{attribute 'qualified_only'}
VAR_GLOBAL
	GC : ARRAY[1..Param_Config.MaxModulePerType] OF FB_GC_Module;
	GC_Runtime : ARRAY[1..Param_Config.MaxModulePerType] OF ST_ModuleRuntimeConfig;
	GC_Control : ARRAY[1..Param_Config.MaxModulePerType] OF ST_GC_CtrlStatus;
	GC_SpinAxis : ARRAY[1..Param_Config.MaxModulePerType] OF I_Axis_BaseUnit;
	GC_LiftPinAxis : ARRAY[1..Param_Config.MaxModulePerType] OF I_Axis_BaseUnit;
END_VAR

(* stored: Version 1.1.0.1, ProductVersion 3.1.4026.18
   GVL GVL_Module: Id {24c37d4f-aefc-4c20-b948-6ed70901060c} *)
